FUNCTION GetComponent : REFERENCE TO Component
VAR_INPUT
	Name: ComponentNames;
END_VAR
VAR
	n: INT;
	Found: int := -1;
	EmptyComponent: Component;
END_VAR

GetComponent REF= EmptyComponent;
FOR n := 0 TO GlobalSettings.MAX_COMPONENTS - 1 DO
	IF GlobalSettings.Components[n].Name = Name THEN
		Found := n;
		EXIT;
	END_IF
END_FOR

IF Found >= 0 THEN
	GetComponent REF= GlobalSettings.Components[Found];
END_IF

END_FUNCTION

(* stored: Version 1.1.0.1, ProductVersion 3.1.4024.6
   POU GetComponent: Id {746cb20f-f503-4212-b9fd-5d00e02fc528}, SpecialFunc None *)
